TYPE T_SimpleStruct : ST_Simple; END_TYPE

(* stored: Version 1.1.0.1
   DUT T_SimpleStruct: Id {0f007a22-d954-4a41-861d-fc41bc28cb8f} *)
